FUNCTION TcoBytesToInt : INT
VAR_INPUT
    inFormat : eTcoDataFormat;
    inByte0 : BYTE;
    inByte1 : BYTE;
END_VAR
VAR
    _b0 : BYTE;
    _b1 : BYTE;
    _tmpWORD : WORD;
END_VAR

IF inFormat = eTcoDataFormat.LittleEndian THEN
    _b0 := inByte1;
    _b1 := inByte0;
ELSIF inFormat = eTcoDataFormat.BigEndian THEN
    _b0 := inByte0;
    _b1 := inByte1;
END_IF

_tmpWORD := _b0;
_tmpWORD := SHL(_tmpWORD, 8);
_tmpWORD := _tmpWORD + _b1;
TcoBytesToInt := WORD_TO_INT(_tmpWORD);

END_FUNCTION

(* stored: Version 1.1.0.1, ProductVersion 3.1.4024.10
   POU TcoBytesToInt: Id {113cf9f7-7deb-4487-9651-4a789b828e1d}, SpecialFunc None *)
